// Application main function
//
PROGRAM MAIN
VAR

	// Function blocks...
	fbHeaterCtrl: FB_HeaterCtrl; // Heater control
	
	// Other members...
	Cntr: DINT; // Counter, visiting times
	Step: SINT; // Step counter (1...100)
	
END_VAR

// Update counter
Cntr := ( Cntr + 1 );

// Hasn't the step counter overflowed yet ?
IF Step < 100 THEN

	// Increase the step counter
	Step := ( Step + 1 );
	
// else, Maximum value reached already
ELSE

	// Restart the step counter
	Step := 1;
	
END_IF

// Call the heater control
fbHeaterCtrl( Step := Step );

// Update history
UpdateHistory( Step );

END_PROGRAM

(* stored: Version 1.1.0.1, ProductVersion 3.1.4022.6
   POU MAIN: Id {6701c937-988a-4712-9161-41d277dbef40}, SpecialFunc None *)
